FUNCTION_BLOCK F_TO_C_CONV (* Template for a Simple Function Block Type *)
  (* Standard: 61499-1 *)
  (* Version 1.0, 2018-12-03, badger *)
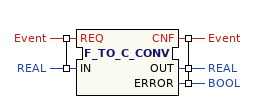
  EVENT_INPUT
    REQ WITH IN; (* Normal Execution Request *)
  END_EVENT
  EVENT_OUTPUT
    CNF WITH OUT, ERROR; (* Execution Confirmation *)
  END_EVENT
  VAR_INPUT
    IN : REAL := 0.00; (* Fahrenheit temperature to be converted *)
  END_VAR
  VAR_OUTPUT
    OUT : REAL := 0.00; (* Converted temperature in celcius *)
    ERROR : BOOL := false; (* Set true when the temperature cannot be converted *)
  END_VAR
  ALGORITHM REQ IN ST: (* Normally executed algorithm *)
	ERROR := FALSE;
	OUT := (IN - 32) * 5 / 9;
	IF (OUT < -273) THEN
		ERROR := TRUE;
	END_IF;
  END_ALGORITHM
END_FUNCTION_BLOCK
